Universal Robots URScript: group.script

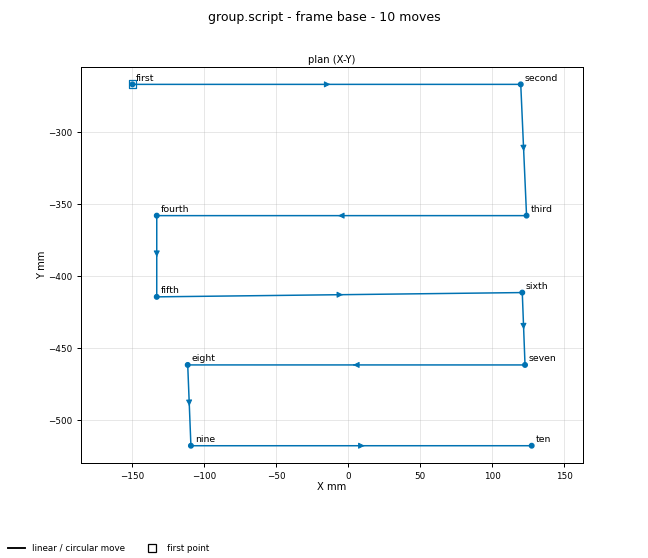
[picture p0: tool path of group.script in frame base, 10 of 10 moves have a stored position in this frame; points joined in program order, loops and branches not executed]
def group():
  global _hidden_verificationVariable=0
  step_count_e284af76_563d_42e6_8820_c6cbdb4f6a84 = 0.0
  thread Step_Counter_Thread_0d8bd874_879c_4191_8d56_159faceed09d():
    while (True):
      step_count_e284af76_563d_42e6_8820_c6cbdb4f6a84 = step_count_e284af76_563d_42e6_8820_c6cbdb4f6a84 + 1.0
      sync()
    end
  end
  run Step_Counter_Thread_0d8bd874_879c_4191_8d56_159faceed09d()
  set_target_payload(0.110000, [-0.015000, -0.005000, -0.003000], [0.000039, 0.000039, 0.000039, 0.000000, 0.000000, 0.000000])
  set_standard_analog_input_domain(0, 1)
  set_standard_analog_input_domain(1, 1)
  set_tool_analog_input_domain(0, 1)
  set_tool_analog_input_domain(1, 1)
  set_analog_outputdomain(0, 0)
  set_analog_outputdomain(1, 0)
  set_input_actions_to_default()
  set_gravity([0.0, 0.0, 9.82])
  set_tcp(p[0.0013207278316754306,-0.005838214497000324,0.07610644847508113,0.0,0.0,0.0])
  set_safety_mode_transition_hardness(1)
  set_tool_communication(False, 115200, 0, 1, 1.5, 3.5)
  set_tool_output_mode(0)
  set_tool_digital_output_mode(0, 1)
  set_tool_digital_output_mode(1, 1)
  set_tool_voltage(0)
  global Plane_1=p[-0.17350531486565687,-0.4033067775546656,0.1772488075736387,1.1232876443030053,0.07343349430999357,0.2514050721194209]
  global WALL=p[-0.29663055217316037,0.3589849393106626,0.09185225943382165,-1.5800000000000005,-0.0015260302561452153,-0.0010686656168337116]
  global belly=p[0.0014478489029917038,-0.32030274011921556,0.1001954744690512,-0.08567825925274844,0.07151626781117665,-1.623822409125042]
  global first_p=p[-.149642120886, -.266701890845, .036436640003, 2.902450510083, -1.202125385623, .000156397430]
  global first_q=[-1.661492172871725, -1.9033752880492152, -2.2266430854797363, -0.5803793233684083, 1.5712440013885498, -2.4413719812976282]
  global second_p=p[.119970548737, -.266696560182, .036421778699, 2.902428888660, -1.202178051423, .000053531278]
  global second_q=[-0.7104571501361292, -1.8468758068480433, -2.319589376449585, -0.5439586204341431, 1.5712778568267822, -1.4900115172015589]
  global third_p=p[.123997428694, -.357852457960, .036428951088, 2.902460618865, -1.202160822920, .000144976257]
  global third_q=[-0.904403034840719, -2.115525861779684, -1.8475925922393799, -0.7472608846477051, 1.5707427263259888, -1.6855924765216272]
  global fourth_p=p[-.132799243417, -.357858271721, .036432259042, 2.902453144836, -1.202139971218, .000174564638]
  global fourth_q=[-1.5933125654803675, -2.1352244816222132, -1.810591220855713, -0.7645800870708008, 1.5707718133926392, -2.374652687703268]
  global fifth_p=p[-.132809259641, -.414252137583, .036436112144, 2.902440175378, -1.202151317604, .000158194687]
  global fifth_q=[-1.5898178259478968, -2.3082028828062953, -1.4775313138961792, -0.9246564668468018, 1.5704803466796875, -2.372479263936178]
  global sixth_p=p[.121030595864, -.411279446985, .036446254016, -2.902440842145, 1.202165496676, -.000291981956]
  global sixth_q=[-0.9915016333209437, -2.276689191857809, -1.5391415357589722, -0.8945059937289734, 1.5705862045288086, -1.773900334035055]
  global seven_p=p[.122935836007, -.461538153955, .036460310453, 2.902467680124, -1.202091376063, .000355998681]
  global seven_q=[-1.047422234212057, -2.4560090504088343, -1.1839351654052734, -1.070316807632782, 1.5703003406524658, -1.8313773314105433]
  global eight_p=p[-.111299028013, -.461523738856, .036442835288, 2.902482438484, -1.202127249959, .000143064515]
  global eight_q=[-1.540938679371969, -2.4545604191222132, -1.1868643760681152, -1.068991021519043, 1.570274829864502, -2.3248634974109095]
  global nine_p=p[-.109074138714, -.517643529543, .036440145747, 2.902494020624, -1.202134298515, .000202157994]
  global nine_q=[-1.5385039488421839, -2.729706426660055, -0.6253552436828613, -1.3553463977626343, 1.5699762105941772, -2.324918810521261]
  global ten_p=p[.127572071405, -.517631146121, .036417220472, -2.902476683840, 1.202061636237, -.000131787598]
  global ten_q=[-1.0925386587726038, -2.7430879078307093, -0.5977126955986023, -1.3696239751628418, 1.5699315071105957, -1.879115406666891]
  while (True):
    $ 2 "Robot Program"
    $ 3 "MoveL"
    $ 4 "first" "breakAfter"
    movel(first_p, a=1.2, v=0.25)
    $ 5 "second" "breakAfter"
    movel(second_p, a=1.2, v=0.25)
    $ 6 "third" "breakAfter"
    movel(third_p, a=1.2, v=0.25)
    $ 7 "fourth" "breakAfter"
    movel(fourth_p, a=1.2, v=0.25)
    $ 8 "fifth" "breakAfter"
    movel(fifth_p, a=1.2, v=0.25)
    $ 9 "sixth" "breakAfter"
    movel(sixth_p, a=1.2, v=0.25)
    $ 10 "seven" "breakAfter"
    movel(seven_p, a=1.2, v=0.25)
    $ 11 "eight" "breakAfter"
    movel(eight_p, a=1.2, v=0.25)
    $ 12 "nine" "breakAfter"
    movel(nine_p, a=1.2, v=0.25)
    $ 13 "ten" "breakAfter"
    movel(ten_p, a=1.2, v=0.25)
  end
end
